(* Schneider Machine Expert - Basic project example1, file version 1.9.0.0 *)
(* ProjectInformations: Name=New project *)

HARDWARE
  Cpu 0: TM221M16R/G
  EthernetConfiguration: NetworkName=M221, IpAllocationMode=FixedAddress, IpAddress=0.0.0.0, SubnetMask=0.0.0.0
  SerialLineConfiguration: Baud=Baud19200, Parity=ParityEven, DataBits=DataBits8, StopBits=StopBits1, PhysicalMedium=PhysicalMediumRs485, TransmissionMode=TransmissionModeModbusRtu, SlaveId=1, Addressing=SlaveAddressing
  MastTask: UsePeriodScanMode=false, PeriodScan=100
  FastTask: Period=255
  CpuBehavior: StartingMode=StartAsPreviousState, AutoSaveRamOnEeprom=true, WatchdogPeriod=250

SYMBOLS  (address, symbol, comment, settings)
  %M10      MEM10  "__NOT__"
  %TM0        [Type=TP, Preset=3, Base=OneSecond]
  %TM1        [Type=TP, Preset=5, Base=OneSecond]
  %I0.0     B_INPUT
  %I0.1     G_INPUT  "__NOT__"
  %Q0.0     B_OUTPUT
  %Q0.1     G_OUTPUT  "__NOT__"

POU New POU
  (* SectionNumber=1 *)

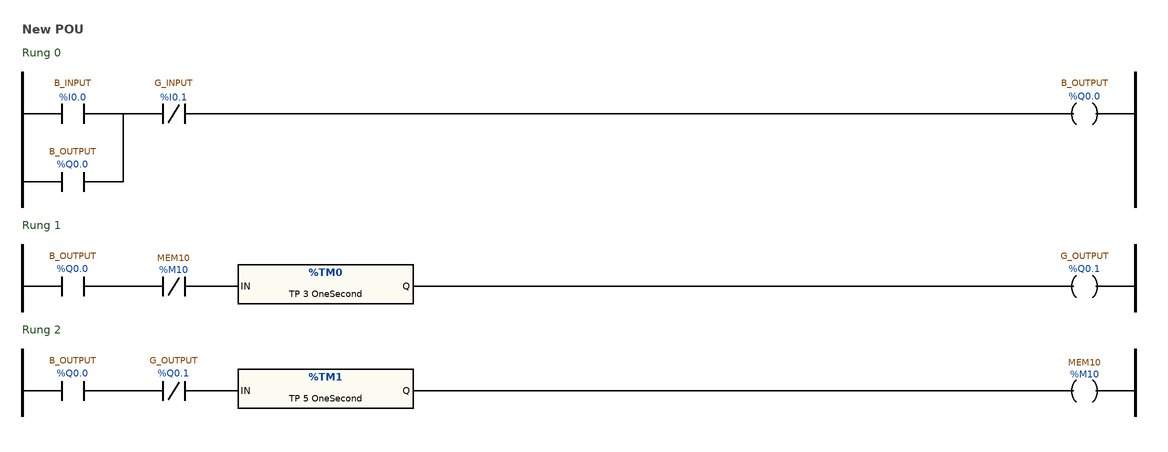

// Rung 0
  LD %I0.0                (* B_INPUT *)
  OR %Q0.0                (* B_OUTPUT *)
  ANDN %I0.1              (* G_INPUT *)
  ST %Q0.0                (* B_OUTPUT *)
  // as ST:
  //   B_OUTPUT := (B_INPUT OR B_OUTPUT) AND NOT G_INPUT;

// Rung 1
  BLK %TM0
  LD %Q0.0                (* B_OUTPUT *)
  ANDN %M10               (* MEM10 *)
  IN
  OUT_BLK
  LD Q
  ST %Q0.1                (* G_OUTPUT *)
  END_BLK
  // as ST:
  //   %TM0(IN := B_OUTPUT AND NOT MEM10);
  //   G_OUTPUT := %TM0.Q;

// Rung 2
  BLK %TM1
  LD %Q0.0                (* B_OUTPUT *)
  ANDN %Q0.1              (* G_OUTPUT *)
  IN
  OUT_BLK
  LD Q
  ST %M10                 (* MEM10 *)
  END_BLK
  // as ST:
  //   %TM1(IN := B_OUTPUT AND NOT G_OUTPUT);
  //   MEM10 := %TM1.Q;
